TYPE ST_TableNumberIn :
STRUCT
END_STRUCT
END_TYPE

(* stored: Version 1.1.0.1
   DUT ST_TableNumberIn: Id {9829719d-0ea9-0cb6-2aa5-9de993fb44b6} *)
